# EPICS StreamDevice protocol: TC110App/Db/TC110.proto
Terminator = CR;

#002 Standby
readStandby {out "0010000202=?%+<sum8>";in "0011000206%6d%+<sum8>";}
setStandby {out "0011000206%{000000|111111}%+<sum8>";in "0011000206%6d%+<sum8>";}

#010 Pumping station
readPumpgStatn {out "0010001002=?%+<sum8>";in "0011001006%6d%+<sum8>";}
setPumpgStatn {out "0011001006%{000000|111111}%+<sum8>";in "0011001006%6d%+<sum8>";}

#012 Enable venting
readenablevent {out "0010001202=?%+<sum8>";in "0011001206%6d%+<sum8>";}
setenablevent {out "0011001206%{000000|111111}%+<sum8>";in "0011001206%6d%+<sum8>";}

#023 Motor Pump
readmotorpump {out "0010002302=?%+<sum8>";in "0011002306%6d%+<sum8>";}
setmotorpump {out "0011002306%{000000|111111}%+<sum8>";in "0011002306%6d%+<sum8>";}

#025 Operation mode backing pump
readOpModeBKP {out "0010002502=?%+<sum8>";in "0011002503%3d%+<sum8>";}
setOpModeBKP {out "0011002503%3.3d%+<sum8>";in "0011002503%3d%+<sum8>";}

#026 Rotation speed setting mode
readSpdSetMode {out "0010002602=?%+<sum8>";in "0011002603%3d%+<sum8>";}
setSpdSetMode {out "0011002603%3.3d%+<sum8>";in "0011002603%3d%+<sum8>";}

#027 gas mode
readgasmode {out "0010002702=?%+<sum8>";in "0011002703%3d%+<sum8>";}
setgasmode {out "0011002703%3.3d%+<sum8>";in "0011002703%3d%+<sum8>";}

#030 Venting mode
readventingmode {out "0010003002=?%+<sum8>";in "0011003003%3d%+<sum8>";}
setventingmode {out "0011003003%3.3d%+<sum8>";in "0011003003%3d%+<sum8>";}

#326 Temperature electronics
readTempElec {out "0010032602=?%+<sum8>"; in "0011032606%6d%+<sum8>";}

#397 Actual rotation speed
readsetRotSpdrpm {out "0010039702=?%+<sum8>"; in "0011039706%6d%+<sum8>";}

#398 Actual rotation speed
readActualSpdrpm {out "0010039802=?%+<sum8>"; in "0011039806%6d%+<sum8>";}

#707 rotation speed setting mode
readSpdSVal {out "0010070702=?%+<sum8>";in "0011070706%6d%+<sum8>";}
setSpdSVal {out "0011070706%6.6d%+<sum8>";in "0011070706%6d%+<sum8>";}

#717 set rotation speed at standby
readSpdbySVal {out "0010071702=?%+<sum8>";in "0011071706%6d%+<sum8>";}
setSpdbySVal {out "0011071706%6.6d%+<sum8>";in "0011071706%6d%+<sum8>";}

#720 Vent speed
readVentSpd {out "0010072002=?%+<sum8>";in "0011072003%3d%+<sum8>";}
setVentSpd {out "0011072003%3.3d%+<sum8>";in "0011072003%3d%+<sum8>";}

#721 Vent time
readVentTime {out "0010072102=?%+<sum8>";in "0011072106%6d%+<sum8>";}
setVentTime {out "0011072106%6.6d%+<sum8>";in "0011072106%6d%+<sum8>"}
